FUNCTION_BLOCK overcurrent (* Template for a simple Basic Function Block Type *)
  (* Standard: 61499-2 *)
  (* Version 1.0, 2021-02-27, badger *)
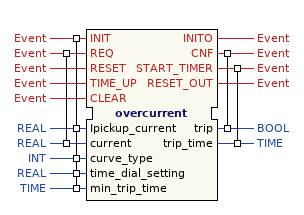
  EVENT_INPUT
    INIT WITH Ipickup_current, curve_type, time_dial_setting, min_trip_time; (* Initialization Request *)
    REQ WITH current; (* Normal Execution Request *)
    RESET;
    TIME_UP;
    CLEAR;
  END_EVENT
  EVENT_OUTPUT
    INITO; (* Initialization Confirm *)
    CNF WITH trip; (* Execution Confirmation *)
    START_TIMER WITH trip_time;
    RESET_OUT;
  END_EVENT
  VAR_INPUT
    Ipickup_current : REAL; (* Input event qualifier *)
    current : REAL;
    curve_type : INT;
    time_dial_setting : REAL;
    min_trip_time : TIME;
  END_VAR
  VAR_OUTPUT
    trip : BOOL; (* Output event qualifier *)
    trip_time : TIME;
  END_VAR
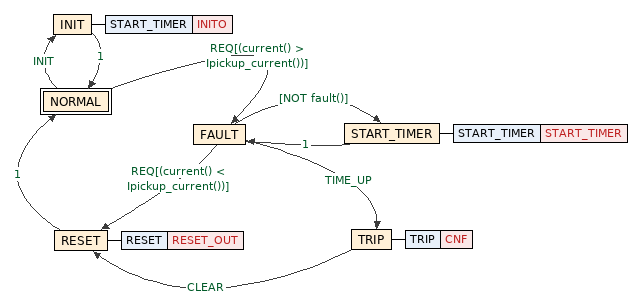
  EC_STATES
    NORMAL; (* Initial State *)
    INIT : START_TIMER -> INITO; (* Initialization *)
    FAULT;
    START_TIMER : START_TIMER -> START_TIMER;
    TRIP : TRIP -> CNF;
    RESET : RESET -> RESET_OUT;
  END_STATES
  EC_TRANSITIONS
    NORMAL TO INIT := INIT;
    INIT TO NORMAL := 1; (* Return after initialisation *)
    NORMAL TO FAULT := REQ[(current() > Ipickup_current())]; (* Starts the timer when an overcurrent fault is detected *)
    FAULT TO START_TIMER := [NOT fault()]; (* Start the time on a fault condition only if it has not already been started. *)
    START_TIMER TO FAULT := 1;
    FAULT TO TRIP := TIME_UP; (* Timer has expired during a fault, signaling that the fault is real. *)
    FAULT TO RESET := REQ[(current() < Ipickup_current())]; (* Clear the fault condition if the current returns to a safe level. *)
    RESET TO NORMAL := 1;
    TRIP TO RESET := CLEAR; (* Stop the time and reset if the fault condition has been cleared. *)
  END_TRANSITIONS
  ALGORITHM INIT IN AnyText: (* Initialisation *)
fault() = false;
  END_ALGORITHM
  ALGORITHM START_TIMER IN AnyText: (* Start timer *)
	fault() = true;
	trip_time() = min_trip_time()
  END_ALGORITHM
  ALGORITHM RESET IN AnyText: (* Reset to clear the fault condition *)
	fault() = false;
  END_ALGORITHM
  ALGORITHM TRIP IN AnyText: (* Trip the circuit breaker *)

  END_ALGORITHM
END_FUNCTION_BLOCK
